// TIA Portal V16 export
// export: Created 2021-09-08T12:46:10.0961874Z, ExportSetting WithDefaults, DisplayName Totally Integrated Automation Portal, DisplayVersion V16 Update 3, DisplayName TIA Portal Version Control Interface, DisplayVersion V16 Update 2, DisplayName TIA Portal Openness, DisplayVersion V16 Update 3, DisplayName TIA Portal Teamcenter Gateway, DisplayVersion V16, DisplayName STEP 7 Professional, DisplayVersion V16 Update 3, DisplayName STEP 7 Safety, DisplayVersion V16, DisplayName WinCC Advanced, DisplayVersion V16 Update 3
FUNCTION_BLOCK "DevBlockAckSingleAlarm"   // FB55, LAD
{ S7_Optimized_Access := 'TRUE' }
VERSION : 0.1
// stored: AutoNumber true, IsIECCheckEnabled false, IsRetainMemResEnabled false, MemoryReserve 100, SetENOAutomatically false, UDAEnableTagReadback false
   VAR_INPUT
      ack : Bool;
   END_VAR
   VAR_IN_OUT
      alarmSignal : Bool;
      ackBit : Bool;
      stateBit : Bool;
      alarmTag : Bool;
   END_VAR
   VAR
      ACK_TAG : TON_TIME;
   END_VAR
   VAR CONSTANT
      ACK_DELAY : Time := T#2s;
   END_VAR
BEGIN

REGION Network 1
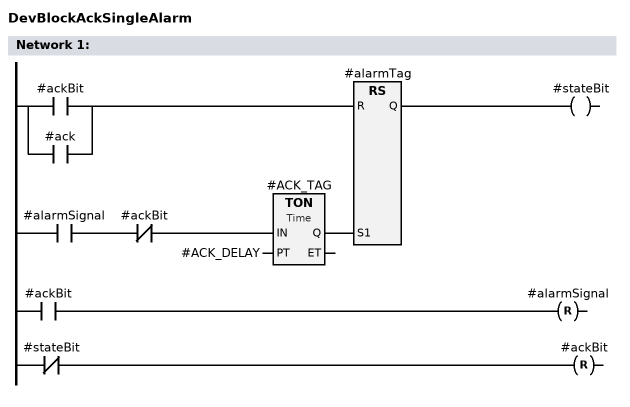
   RUNG wire#powerrail
      Contact( #ackBit )
      wire#w1
      S_RS(operand := #alarmTag, s1 := wire#w2)
      Coil( #stateBit )
   END_RUNG
   RUNG wire#powerrail
      Contact( #ack )
   END_RUNG wire#w1
   RUNG wire#powerrail
      Contact( #alarmSignal )
      I_Contact( #ackBit )
      { S7_Templates := "time_type := Time" } #ACK_TAG.TON(pt := #ACK_DELAY, et =>)
   END_RUNG wire#w2
   RUNG wire#powerrail
      Contact( #ackBit )
      R_Coil( #alarmSignal )
   END_RUNG
   RUNG wire#powerrail
      I_Contact( #stateBit )
      R_Coil( #ackBit )
   END_RUNG
   // the same network as SCL:
   #ACK_TAG(IN := #alarmSignal AND NOT #ackBit, PT := #ACK_DELAY);   // TON
   IF #ackBit OR #ack THEN
       #alarmTag := FALSE;   // RS flip-flop
   END_IF;
   IF #ACK_TAG.Q THEN #alarmTag := TRUE; END_IF;
   #stateBit := #alarmTag;
   IF #ackBit THEN #alarmSignal := FALSE; END_IF;
   IF NOT #stateBit THEN #ackBit := FALSE; END_IF;
END_REGION
END_FUNCTION_BLOCK
